// TwinCAT 3 PLC project Untitled1
// ProgramVersion: 3.1.4026.16
// libraries:
//   Tc2_Standard, * (Beckhoff Automation GmbH)
//   Tc2_System, * (Beckhoff Automation GmbH)
// project tree:
//   DUTs/ Space.TcDUT, Weight.TcDUT
//   / PlcTask.TcTTO
//   POUs/ MAIN.TcPOU, ShelfManager.TcPOU, Tests.TcPOU
// real-time tasks:
//   TASK PlcTask: cycle T#10ms, priority 20, ADS port 350

CONFIGURATION Untitled1
    RESOURCE PLC ON TwinCAT3
        TASK PlcTask(INTERVAL := T#10ms, PRIORITY := 20);
        PROGRAM MAIN WITH PlcTask : MAIN;
    END_RESOURCE
END_CONFIGURATION

// ---- DUTs/Space.TcDUT
TYPE Space :
STRUCT
	Column : SINT;
	Row : SINT;
	PartID : STRING;
	Weight : Weight;
END_STRUCT
END_TYPE

// ---- DUTs/Weight.TcDUT
TYPE Weight : (Empty, Light, Heavy);
END_TYPE;

// ---- POUs/MAIN.TcPOU
PROGRAM MAIN
VAR
		
	manager : ShelfManager;
	Reset : BOOL;
	FuncTest : USINT;
	space : Space;
	
	ErrorSameID : BOOL;
	ErrorNotEnoghPlace : BOOL;
	ErrorNothingToBeTakenOut : BOOL;
	ErrorNotFound : BOOL;
	ErrorCantStoreWithoutProperties : BOOL;
	ErrorSerchWithoutPartID : BOOL;
	ErrorSpaceDoesNotExist : BOOL;
	
	doTests : BOOL;
	tests : Tests;
	
END_VAR

manager(
	ErrorNotFound => ErrorNotFound,
	ErrorSameID => ErrorSameID,
	ErrorNothingToBeTakenOut => ErrorNothingToBeTakenOut,
	ErrorNothingToBeTakenOut => ErrorNothingToBeTakenOut,
	ErrorReset := Reset,
	ErrorCantStoreWithoutProperties => ErrorCantStoreWithoutProperties,
	ErrorSerchWithoutPartID => ErrorSerchWithoutPartID,
	ErrorSpaceDoesNotExist => ErrorSpaceDoesNotExist
);

CASE FuncTest OF
	1:
		manager.FindPart(
			SerchingPartID := space.PartID,
			FoundPart => space
		);	
	2:
		space := manager.NextFreeSpaceLight;	
	3:
		space := manager.NextFreeSpaceHeavy;
	4: 
		space := manager.NextOccupiedSpace;
	5:
	 	manager.RemoveByID(removedPartID := space.PartID);
	6: 
		manager.RemoveFIFO();
	7:
		manager.RemoveExplicit(
			column := (space.Column),
			row := (space.Row)
		);	
	8: 
		manager.StoreFIFO(
			storedFifoID := space.PartID,
			storedFifoWeight := space.Weight
		);
	9: 
		manager.StoreExplicit(storedPart := space);
	
END_CASE
FuncTest := 0;

IF doTests THEN
	tests();
	doTests := FALSE;
END_IF

END_PROGRAM

// ---- POUs/ShelfManager.TcPOU
FUNCTION_BLOCK ShelfManager
VAR_INPUT
	ErrorReset : BOOL;
END_VAR
VAR_OUTPUT
	ErrorSameID : BOOL;
	ErrorNotEnoghPlace : BOOL;
	ErrorNothingToBeTakenOut : BOOL;
	ErrorNotFound : BOOL;
	ErrorCantStoreWithoutProperties : BOOL;
	ErrorSerchWithoutPartID : BOOL;
	ErrorSpaceDoesNotExist : BOOL;
END_VAR
VAR CONSTANT
	NOFSPACES : SINT := 42;
	NOFCOLUMNS : SINT := 7;
	NOFROWS : SINT := 6;
END_VAR
VAR
	initialized : BOOL;
	x : SINT;
	y : SINT;
	Z : SINT;
	Spaces : ARRAY [0..NOFSPACES - 1] OF Space;	
END_VAR

IF NOT initialized THEN
	FOR x := 0 TO (NOFROWS - 1) DO
		FOR y := 0 TO (NOFCOLUMNS - 1) DO
			Spaces[Z].Column := y;
			Spaces[Z].Row := x;
			Spaces[Z].partID := '';
			Spaces[Z].Weight := Empty;
			Z := Z + 1;
		END_FOR

	END_FOR
	initialized := TRUE;
END_IF


IF ErrorReset THEN
	ErrorSameID := FALSE;
	ErrorNotEnoghPlace := FALSE;
	ErrorNothingToBeTakenOut := FALSE;
	ErrorNotFound := FALSE;
	ErrorCantStoreWithoutProperties := FALSE;
	ErrorSerchWithoutPartID := FALSE;
	ErrorSpaceDoesNotExist := FALSe;
END_IF

METHOD FindPart : BOOL;
VAR_INPUT
	SerchingPartID	: STRING;
END_VAR
VAR_OUTPUT
	FoundPart : Space;
END_VAR
FindPart := FALSE;
IF (SerchingPartID = '') THEN
	ErrorSerchWithoutPartID := TRUE;
	RETURN;
END_IF;

FOR x := 0 TO (NOFSPACES - 1) DO
	IF Spaces[x].partID = SerchingPartID  THEN
		FoundPart := Spaces[x];
		FindPart := TRUE;
		RETURN;
	END_IF
	IF x = (NOFSPACES - 1) THEN
		FindPart := FALSE;
		RETURN;
	END_IF
END_FOR
END_METHOD

PROPERTY NextFreeSpaceHeavy : Space
GET
VAR
	n : SINT;
	y : SINT;
	actNextFree : Space;
END_VAR
actNextFree.Column := -1;

FOR y := 0 TO NOFROWS - 1 DO
	FOR n := 0 TO NOFSPACES - 1 DO
		IF Spaces[n].Row = y AND Spaces[n].PartID = '' AND Spaces[n].Column	> actNextFree.Column THEN
			actNextFree := Spaces[n];
		END_IF
	END_FOR
	IF NOT (actNextFree.Column = -1) THEN
		NextFreeSpaceHeavy := actNextFree;
		RETURN;
	END_IF
END_FOR

ErrorNotEnoghPlace := TRUE;
END_GET
END_PROPERTY

PROPERTY NextFreeSpaceLight : Space
GET
VAR
	n : SINT;
	y : SINT;
	actNextFree : Space;
END_VAR
actNextFree.Column := NOFCOLUMNS;

FOR y := NOFROWS - 1 TO 0 BY -1 DO
	FOR n := 0 TO NOFSPACES - 1 DO
		IF Spaces[n].Row = y AND Spaces[n].PartID = '' AND Spaces[n].Column	< actNextFree.Column THEN
			actNextFree := Spaces[n];
		END_IF
	END_FOR
	IF NOT (actNextFree.Column = NOFCOLUMNS) THEN
		NextFreeSpaceLight := actNextFree;
		RETURN;
	END_IF
END_FOR

ErrorNotEnoghPlace := TRUE;
END_GET
END_PROPERTY

PROPERTY NextOccupiedSpace : Space
GET
FOR x := 0 TO (NOFSPACES - 1) DO
	IF NOT (Spaces[x].partID = '') THEN
		NextOccupiedSpace := Spaces[x];
		RETURN;
	ELSIF x = (NOFSPACES - 1) THEN
		ErrorNothingToBeTakenOut := TRUE;	
		RETURN;	
	END_IF
END_FOR
END_GET
END_PROPERTY

METHOD RemoveByID : BOOL
VAR_INPUT
	removedPartID	: STRING;
END_VAR
VAR	
	foundPart : Space;
END_VAR
IF FindPart(SerchingPartID := removedPartID,FoundPart => foundPart)THEN
	RemoveByID := RemoveExplicit(column := foundPart.Column,row := foundPart.Row);
ELSE
	RemoveByID := FALSE;
END_IF
END_METHOD

METHOD RemoveExplicit : BOOL
VAR_INPUT
	Column : SINT;
	Row	: SINT;
END_VAR
VAR
END_VAR
RemoveExplicit := FALSE;

IF (Column < 0 OR Column > 6) OR
   (Row    < 0 OR Row    > 5) THEN
	ErrorSpaceDoesNotExist := TRUE;
	RETURN;
END_IF

FOR x := 0 TO (NOFSPACES - 1) DO
	IF Spaces[x].Column = column AND Spaces[x].Row = row THEN
		IF (Spaces[x].partID = '') THEN
			ErrorNothingToBeTakenOut := TRUE;
			RETURN;
		ELSE
			FOR y := x + 1 TO (NOFSPACES - 1) DO
				Spaces[y-1] := Spaces[y];
			END_FOR
			Spaces[NOFSPACES - 1].Column := column;
			Spaces[NOFSPACES - 1].Row := row;
			Spaces[NOFSPACES - 1].partID := '';
			Spaces[NOFSPACES - 1].Weight := Empty;
			RemoveExplicit := TRUE;
			RETURN;
		END_IF
	END_IF
END_FOR
END_METHOD

METHOD RemoveFIFO : BOOL
VAR_INPUT
END_VAR
VAR	
	removedFifoSpace : Space;
END_VAR
RemoveFIFO := FALSE;

removedFifoSpace := NextOccupiedSpace;
IF ErrorNothingToBeTakenOut THEN
	RETURN;
END_IF

RemoveFIFO := RemoveExplicit(column := removedFifoSpace.Column, row := removedFifoSpace.Row);
END_METHOD

METHOD StoreExplicit : BOOL
VAR_INPUT
	storedPart : Space;
END_VAR
VAR
END_VAR
StoreExplicit := FALSE;	

IF (storedPart.Column < 0 OR storedPart.Column > 6) OR
   (storedPart.Row    < 0 OR storedPart.Row    > 5) THEN
	ErrorSpaceDoesNotExist := TRUE;
	RETURN;
ELSIF storedPart.partID = '' OR storedPart.Weight = Empty THEN
	ErrorCantStoreWithoutProperties := TRUE;
	RETURN;
ELSIF FindPart(SerchingPartID := storedPart.partID) THEN
	ErrorSameID := TRUE;
	RETURN;
END_IF	

FOR x := 0 TO (NOFSPACES - 1) DO
	IF Spaces[x].Column = storedPart.Column AND Spaces[x].Row = storedPart.Row THEN
		FOR y := x + 1 TO (NOFSPACES - 1) DO
			Spaces[y-1] := Spaces[y];
		END_FOR
		Spaces[(NOFSPACES - 1)] := storedPart;
		StoreExplicit := TRUE;
		RETURN;				
	END_IF
END_FOR
END_METHOD

METHOD StoreFIFO : BOOL
VAR_INPUT
	storedFifoID : STRING;
	storedFifoWeight : Weight;
END_VAR
VAR	
	storeFifoSpace : Space;
END_VAR
StoreFIFO := FALSE;

IF storedFifoWeight = Weight.Heavy THEN
	storeFifoSpace := NextFreeSpaceHeavy;
ELSE
	storeFifoSpace := NextFreeSpaceLight;
END_IF

IF ErrorNotEnoghPlace THEN
	RETURN;
END_IF

storeFifoSpace.PartID := storedFifoID;
storeFifoSpace.Weight := storedFifoWeight;

storeFifoSpace.partID := storedFifoID;

StoreFIFO := StoreExplicit(storedPart := storeFifoSpace);
END_METHOD

END_FUNCTION_BLOCK

// ---- POUs/Tests.TcPOU
FUNCTION_BLOCK Tests
VAR_INPUT
	Manager : ShelfManager;
END_VAR
VAR_OUTPUT
	TestFullStoringExplicit : BOOL;
	TestRemovingExplicit : BOOL;
	TestRemoveAllFifo : BOOL;
	TestStoreFifo : BOOL;

END_VAR
VAR
END_VAR

Manager();
TestFullStoringExplicit := FullStoringExplicit();
TestRemovingExplicit := RemovingExplicit();
TestRemoveAllFifo := RemoveAllFifo();
TestStoreFifo := StoreFifo();

METHOD FullStoringExplicit : BOOL
VAR_INPUT
END_VAR
VAR	
	x : SINT;
	y : SINT;
	z : SINT;
	space : Space;
END_VAR
FullStoringExplicit := FALSE;

FOR x := 0 TO Manager.NOFROWS - 1 DO
	FOR y := 0 TO Manager.NOFCOLUMNS - 1 DO
		z := z+1;
		space.Column := y;
		space.Row := x;
		space.PartID := INT_TO_STRING(z);
		space.Weight := Weight.Light;
		Manager.StoreExplicit(storedPart := space);
	END_FOR	
END_FOR

IF NOT(Manager.Spaces[0].PartID = '1')THEN
	RETURN; 
ELSIF NOT (Manager.Spaces[Manager.NOFSPACES - 1].PartID = INT_TO_STRING(Manager.NOFSPACES)) THEN
	RETURN;
END_IF

FullStoringExplicit := TRUE;
END_METHOD

METHOD RemoveAllFifo : BOOL
VAR_INPUT
END_VAR
VAR
	n : SINT;
END_VAR
RemoveAllFifo := FALSE;

IF NOT TestRemovingExplicit THEN
	RETURN;
END_IF

FOR n := 2 TO Manager.NOFSPACES DO
	IF NOT (Manager.Spaces[0].PartID = SINT_TO_STRING(n)) THEN
		RETURN;
	END_IF
	Manager.RemoveFIFO();
END_FOR

RemoveAllFifo := TRUE;
END_METHOD

METHOD RemovingExplicit : BOOL
RemovingExplicit := FALSE;

IF NOT TestFullStoringExplicit THEN
	RETURN;
END_IF

IF NOT Manager.RemoveExplicit(Column := 0, Row := 0) THEN
	RETURN;
ELSIF NOT (Manager.Spaces[Manager.NOFSPACES - 1].PartID = '') THEN
	RETURN;
ELSIF NOT (Manager.Spaces[0].PartID = '2') THEN
	RETURN;
END_IF

RemovingExplicit := TRUE;
END_METHOD

METHOD StoreFifo : BOOL
VAR_INPUT
END_VAR
VAR
	n : SINT;
	weight : Weight := Light;
END_VAR
StoreFifo := FALSE;

IF NOT TestRemoveAllFifo THEN
	RETURN;
END_IF

FOR n := 0 TO Manager.NOFSPACES DO
	IF weight = Light THEN
		weight := Heavy;
	ELSE 
		weight := Light;
	END_IF
	Manager.StoreFIFO(
		storedFifoID := SINT_TO_STRING(n),
		storedFifoWeight := weight
	);
END_FOR

IF NOT Manager.ErrorNotEnoghPlace THEN
	RETURN;
END_IF

StoreFifo := TRUE;
END_METHOD

END_FUNCTION_BLOCK
